(* PLC project control_valve_32, Dassault Systèmes ControlBuild 2024x *)
(* stored: creationDateTime 2023-10-03T11:13:12-01:00 *)

(* This module simulates a three-way, two positions control valve used to drive a single-acting jack. *)
FUNCTION_BLOCK equipment_library.control_valve_32
  VAR_INPUT
    energy : BOOL := true;
    cmdSupply : BOOL := true;
  END_VAR
  VAR_INPUT
    ctrlValve : BOOL := false;
  END_VAR
  VAR_OUTPUT
    pipeWork : BOOL := false;
    pipeRest : BOOL := false;
  END_VAR
  VAR_OUTPUT
    workingMode : BOOL := false;
  END_VAR
  VAR
    slidePosition : DINT := 0;
  END_VAR
  VAR
    d_work : BOOL := false;
    v_d_work : BOOL := false;
  END_VAR


ACTION C_source_code:
/* ----------------------------------------------------------------	*/
/* Type : Model of Operative Behaviour					*/
/* Category :  Pre-actuators						*/
/* Author : Dassault Systemes						*/
/* Update date : June 2018							*/
/* ----------------------------------------------------------------	*/
/* This module simulates a three-way, two positions control valve	*/
/* used to drive a single-acting jack.					*/
/* ----------------------------------------------------------------	*/
 
/* ----------------------------------------------------------------	*/
/* Management of orders from Control Part					*/
/*	if there is no power supply for command the solenoid 		*/
/*     control valve doesn't understand the control order.		*/
/* ----------------------------------------------------------------	*/
if (cmdSupply && ctrlValve) {
	slidePosition = 1;
	workingMode=1;
}
else {
	slidePosition = 0;
	workingMode=0;
}

/* ----------------------------------------------------------------	*/
/* Calculation of the on-state of the energy in the pipes		*/
/*     if a fault is required on a pipe, the latter 			*/
/*		 takes a preset state.					*/
/*     if there is no energy in input, pipes are not 			*/
/*	   under pressure.							*/
/* ----------------------------------------------------------------	*/
if (d_work)
	pipeWork = v_d_work;
else
	pipeWork = (slidePosition==1) & energy;
END_ACTION
END_FUNCTION_BLOCK
